Yaskawa INFORM job: R1_W09,10(-70,-90).JBI

/JOB
//NAME R1_W09,10(-70,-90)
///FOLDERNAME KRIS-SCIANA
//POS
///NPOS 90,90,0,3,0,0
///TOOL 0
///POSTYPE PULSE
///PULSE
C00000=105507,6353,10355,32210,77694,10852
C00001=105510,16911,37473,33972,68168,7953
C00002=106445,24038,48124,34610,65395,7429
C00003=106810,27178,52792,34925,64209,7178
C00004=107223,29077,55924,35176,63262,7024
C00005=106810,27178,52792,34925,64209,7178
C00006=111597,34374,55261,24752,67857,12527
C00007=111403,36775,57527,24785,67766,12433
C00008=111597,34374,55261,24752,67857,12527
C00009=105332,23712,52918,45890,61741,2450
C00010=106112,24999,56308,46457,60360,2116
C00011=105309,25689,57724,46644,60385,1721
C00012=106112,24999,56308,46457,60360,2116
C00013=105332,23712,52918,45890,61741,2450
C00014=101707,26902,59274,46629,61886,710
C00015=101134,23494,54458,46158,63013,1015
C00016=99660,15811,43609,45197,65663,1627
C00017=99658,2699,13820,42409,74184,5482
C00018=100944,-23463,-28347,-16970,63480,36977
C00019=108394,-17548,-16019,-49865,70025,-52116
C00020=108398,-10140,6791,-53180,63488,-48177
C00021=106775,-6629,13409,-53973,61180,-47615
C00022=106133,-5117,16180,-54336,60255,-47371
C00023=107291,-5715,15632,-54404,60933,-47123
C00024=107480,-3600,18285,-54658,60715,-46850
C00025=107291,-5715,15632,-54404,60933,-47123
C00026=106133,-5117,16180,-54336,60255,-47371
C00027=112577,-6253,41430,-93353,55998,-31307
C00028=111384,-5852,41817,-93833,55239,-31278
C00029=112577,-6253,41430,-93353,55998,-31307
C00030=112686,-4721,41124,-92655,56052,-31846
C00031=106463,49428,59370,-45801,86010,-53564
C00032=104350,55811,67904,-46166,83549,-53412
C00033=104237,54632,67536,-46206,83224,-53314
C00034=104350,55811,67904,-46166,83549,-53412
C00035=106463,49428,59370,-45801,86010,-53564
C00036=107409,43305,52302,-45656,87343,-53733
C00037=107406,34453,25894,-46161,95648,-57567
C00038=100944,-23463,-28347,-16970,63480,36977
C00039=94322,-8961,4340,58896,67729,20033
C00040=94324,3408,32592,63285,62150,15207
C00041=96015,10228,41945,64521,60078,14442
C00042=93624,22146,60527,72923,62585,13290
C00043=96036,13458,45397,64761,59856,14226
C00044=96779,10789,43766,65030,59240,14171
C00045=93432,22237,60777,72930,62669,13216
C00046=89655,31401,78083,74739,63139,9922
C00047=89612,30497,77324,74727,63164,9920
C00048=88840,27323,72343,73814,64052,10548
C00049=86751,18668,60154,71910,66292,11794
C00050=108533,5227,38528,60264,34879,9720
C00051=109025,14257,49498,62900,33542,8368
C00052=109212,18153,54326,64197,32978,7705
C00053=109686,18455,55784,65177,32363,7265
C00054=109077,15251,50965,63423,33325,8096
C00055=105202,21598,61212,68001,34306,4940
C00056=104958,17433,55991,66572,34891,5673
C00057=104319,7935,44326,63709,36290,7140
C00058=86556,22142,44402,65204,52764,8391
C00059=87809,30735,55573,66950,50921,7317
C00060=88292,34520,60553,67806,50159,6792
C00061=87967,31574,56914,67246,50659,7132
C00062=88137,35000,62373,68477,49910,6289
C00063=97118,24725,50761,66913,45010,8892
C00064=96354,26018,55370,74307,44828,8922
C00065=93966,23196,51689,73389,46630,9096
C00066=91617,16448,42442,71368,48895,10062
C00067=84171,12138,20476,64082,58354,14713
C00068=100944,-23463,-28347,-16970,63480,36977
C00069=96447,22959,14619,-11970,61601,42404
C00070=96448,30386,38961,-13596,50700,43735
C00071=95000,36478,48363,-13431,47877,43489
C00072=94352,38607,52133,-13372,46577,43380
C00073=94243,36562,48804,-13107,47533,43194
C00074=95182,38097,51286,-13726,46966,43705
C00075=93219,32606,51589,-13417,43719,43279
C00076=93740,30628,48635,-13498,44583,43392
C00077=95235,24197,39000,-13662,47382,43668
C00078=96470,6726,37236,-20140,22006,50250
C00079=94871,14470,47044,-19652,19703,49810
C00080=94306,17297,50884,-19635,18719,49724
C00081=93961,15075,48142,-18563,19160,49171
C00082=95170,16994,50557,-20973,18958,50474
C00083=93554,20903,63156,-25970,13231,52537
C00084=93958,18529,59827,-25342,14110,52319
C00085=95585,9687,48585,-24724,16711,52290
C00086=95583,-6925,15414,-14891,27959,47573
C00087=95583,-6925,2254,-14891,27959,47573
C00088=39529,58299,19798,-2800,57622,-12215
C00089=-21926,113881,9055,11361,100142,-74952
BC00000=262825,1112298,947777
BC00001=262825,1112298,947777
BC00002=262825,1112298,947777
BC00003=262825,1112298,947777
BC00004=262825,1112298,947777
BC00005=262825,1112298,947777
BC00006=262825,1112298,947777
BC00007=262825,1112298,947777
BC00008=262825,1112298,947777
BC00009=262825,1112298,947777
BC00010=262825,1112298,947777
BC00011=262825,1112298,947777
BC00012=262825,1112298,947777
BC00013=262825,1112298,947777
BC00014=262825,1112298,947777
BC00015=262825,1112298,947777
BC00016=262825,1112298,947777
BC00017=262825,1112298,947777
BC00018=221705,1109915,813763
BC00019=258119,1070108,850270
BC00020=258119,1070108,850270
BC00021=258119,1070108,850270
BC00022=258119,1070108,850270
BC00023=258119,1070108,850270
BC00024=258119,1070108,850270
BC00025=258119,1070108,850270
BC00026=258119,1070108,850270
BC00027=258119,1070108,850270
BC00028=258119,1070108,850270
BC00029=258119,1070108,850270
BC00030=258119,1070108,850270
BC00031=258119,1070108,850270
BC00032=258119,1070108,850270
BC00033=258119,1070108,850270
BC00034=258119,1070108,850270
BC00035=258119,1070108,850270
BC00036=258119,1070108,850270
BC00037=258119,1070108,850270
BC00038=221705,1109915,813763
BC00039=264373,1115318,867124
BC00040=264373,1115318,867124
BC00041=264373,1115318,867124
BC00042=264373,1115318,867124
BC00043=264373,1115318,867124
BC00044=264373,1115318,867124
BC00045=264373,1115318,867124
BC00046=264373,1115318,867124
BC00047=264373,1115318,867124
BC00048=264373,1115318,867124
BC00049=264373,1115318,867124
BC00050=254240,1140306,907810
BC00051=254240,1140306,907810
BC00052=254240,1140306,907810
BC00053=254240,1140306,907810
BC00054=254240,1140306,907810
BC00055=254240,1140306,907810
BC00056=254240,1140306,907810
BC00057=254240,1140306,907810
BC00058=202332,1150246,830066
BC00059=202332,1150246,830066
BC00060=202332,1150246,830066
BC00061=202332,1150246,830066
BC00062=202332,1150246,830066
BC00063=202332,1150246,830066
BC00064=202332,1150246,830066
BC00065=202332,1150246,830066
BC00066=202332,1150246,830066
BC00067=202332,1150246,830066
BC00068=221705,1109915,813763
BC00069=254414,1120928,900171
BC00070=254414,1120928,900171
BC00071=254414,1120928,900171
BC00072=254414,1120928,900171
BC00073=254414,1120928,900171
BC00074=254414,1120928,900171
BC00075=254414,1120928,900171
BC00076=254414,1120928,900171
BC00077=254414,1120928,900171
BC00078=263722,1123674,907456
BC00079=263722,1123674,907456
BC00080=263722,1123674,907456
BC00081=263722,1123674,907456
BC00082=263722,1123674,907456
BC00083=263722,1123674,907456
BC00084=263722,1123674,907456
BC00085=263722,1123674,907456
BC00086=263722,1123674,907456
BC00087=263722,1123674,907456
BC00088=202285,940925,986430
BC00089=86457,701907,1069891
///POSTYPE BASE
///RECTAN
///RCONF 0,0,0,0,0,0,0,0,0,0,0,0,0,0,0,0,0,0,0,0,0,0,0,0
P00006=0.222,-3.123,-1.508,0.0000,0.0000,0.0000
P00021=-0.225,-6.128,-0.405,0.0000,0.0000,0.0000
P00027=-0.746,0.015,-9.096,0.0000,0.0000,0.0000
//INST
///DATE 2024/07/23 15:15
///ATTR SC,RW
///GROUP1 RB1,BS1
NOP
'r1_W09,10(-70,-90)
'Path S790 (for W407)
SFTOF
MOVJ C00000 BC00000 VJ=80.00
MOVJ C00001 BC00001 VJ=80.00
MOVJ C00002 BC00002 VJ=20.00
MOVL C00003 BC00003 V=60.0
REFP 3 C00004 BC00004
CALL JOB:SEARCH-R1
SET P021 P006
SFTON P021
MOVL C00005 BC00005 V=60.0
MOVL C00006 BC00006 V=60.0
REFP 3 C00007 BC00007
CALL JOB:SEARCH-R1
SET P021 P006
SFTON P021
MOVL C00008 BC00008 V=60.0
MOVL C00009 BC00009 V=100.0
MOVL C00010 BC00010 V=60.0
REFP 3 C00011 BC00011
CALL JOB:SEARCH-R1
SET P021 P006
SFTON P021
MOVL C00012 BC00012 V=60.0
MOVL C00013 BC00013 V=100.0
MOVL C00014 BC00014 V=100.0
MOVL C00015 BC00015 V=100.0
MOVL C00016 BC00016 V=166.7
MOVL C00017 BC00017 V=166.7
MOVJ C00018 BC00018 VJ=80.00
'Path S793 (for W410)
SFTOF
MOVJ C00019 BC00019 VJ=100.00
MOVJ C00020 BC00020 VJ=100.00
MOVJ C00021 BC00021 VJ=20.00
MOVL C00022 BC00022 V=100.0
MOVL C00023 BC00023 V=60.0
REFP 3 C00024 BC00024
CALL JOB:SEARCH-R1
SET P027 P006
SFTON P027
MOVL C00025 BC00025 V=60.0
MOVL C00026 BC00026 V=100.0
MOVL C00027 BC00027 V=60.0
REFP 3 C00028 BC00028
CALL JOB:SEARCH-R1
SET P027 P006
SFTON P027
MOVL C00029 BC00029 V=60.0
MOVL C00030 BC00030 V=100.0
MOVL C00031 BC00031 V=100.0
MOVL C00032 BC00032 V=60.0
REFP 3 C00033 BC00033
CALL JOB:SEARCH-R1
SET P027 P006
SFTON P027
MOVL C00034 BC00034 V=60.0
MOVL C00035 BC00035 V=100.0
MOVL C00036 BC00036 V=166.7
MOVL C00037 BC00037 V=166.7
MOVJ C00038 BC00038 VJ=100.00
'Path W407
SFTOF
SFTON P021
MOVJ C00039 BC00039 VJ=100.00
MOVJ C00040 BC00040 VJ=100.00
MOVJ C00041 BC00041 VJ=20.00
MOVL C00042 BC00042 V=100.0 PL=0
REFP 1 C00043 BC00043
REFP 2 C00044 BC00044
MACRO1 MJ#(0) ARGF6
ARCON
MOVL C00045 BC00045 V=10.0
MOVL C00046 BC00046 V=10.0
MOVL C00047 BC00047 V=10.0
ARCOF
MOVL C00048 BC00048 V=100.0
MOVL C00049 BC00049 V=166.7
SFTOF
'Path W408
SFTOF
SFTON P021
MOVJ C00050 BC00050 VJ=20.00
MOVJ C00051 BC00051 VJ=20.00
MOVL C00052 BC00052 V=100.0 PL=0
REFP 1 C00053 BC00053
REFP 2 C00054 BC00054
MACRO1 MJ#(0) ARGF6
ARCON
MOVL C00055 BC00055 V=10.0
ARCOF
MOVL C00056 BC00056 V=100.0
MOVL C00057 BC00057 V=166.7
SFTOF
'Path W409
SFTOF
SFTON P021
MOVJ C00058 BC00058 VJ=50.00
MOVJ C00059 BC00059 VJ=20.00
TIMER T=1.00
MOVL C00060 BC00060 V=100.0 PL=0
REFP 1 C00061 BC00061
REFP 2 C00062 BC00062
MACRO1 MJ#(0) ARGF0
ARCON
MOVL C00063 BC00063 V=8.3
MOVL C00064 BC00064 V=8.3
ARCOF
MOVL C00065 BC00065 V=100.0
MOVL C00066 BC00066 V=166.7
MOVL C00067 BC00067 V=166.7
SFTOF
MOVJ C00068 BC00068 VJ=80.00
'
'Path W410
SFTOF
SFTON P027
MOVJ C00069 BC00069 VJ=100.00
MOVJ C00070 BC00070 VJ=100.00
MOVJ C00071 BC00071 VJ=20.00
MOVL C00072 BC00072 V=100.0 PL=0
REFP 1 C00073 BC00073
REFP 2 C00074 BC00074
MACRO1 MJ#(0) ARGF6
ARCON
MOVL C00075 BC00075 V=8.3
ARCOF
MOVL C00076 BC00076 V=100.0
MOVL C00077 BC00077 V=166.7
SFTOF
'Path W1046
SFTOF
SFTON P027
MOVJ C00078 BC00078 VJ=20.00
MOVJ C00079 BC00079 VJ=20.00
MOVL C00080 BC00080 V=100.0 PL=0
REFP 1 C00081 BC00081
REFP 2 C00082 BC00082
MACRO1 MJ#(0) ARGF6
ARCON
MOVL C00083 BC00083 V=8.3
ARCOF
MOVL C00084 BC00084 V=83.3
MOVL C00085 BC00085 V=83.3
MOVL C00086 BC00086 V=83.3
SFTOF
MOVJ C00087 BC00087 VJ=100.00
MOVJ C00088 BC00088 VJ=100.00
MOVJ C00089 BC00089 VJ=100.00
END
